PROGRAM MAIN
VAR
	TankControl01				: TankControl;
	Enable						: BOOL;
	TempReq						: REAL := 22.0;
	VolReq						: REAL := 1.2;
	TankDiam					: REAL := 1.0;
	TankHeight					: REAL := 10;
	LevelSensor					: WORD;
	TempSensor					: WORD;
	StartControl				: BOOL;
	FillValve					: BOOL;
	EmptyValve					: BOOL;
	HeatValve					: BOOL;
	
	Temp						: REAL;
	MixerMotor: BOOL;
END_VAR

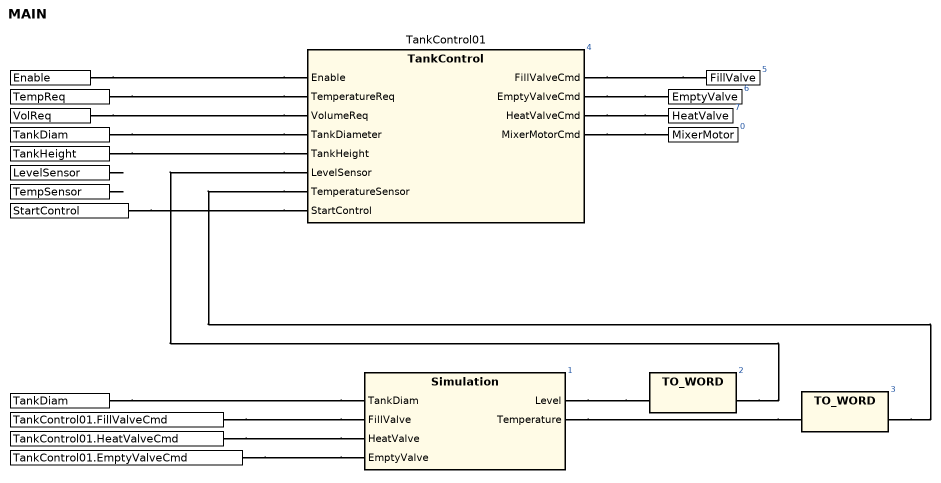
MixerMotor := TankControl01.MixerMotorCmd;
Simulation(TankDiam := TankDiam, FillValve := TankControl01.FillValveCmd, HeatValve := TankControl01.HeatValveCmd, EmptyValve := TankControl01.EmptyValveCmd);
TankControl01(
    Enable := Enable,
    TemperatureReq := TempReq,
    VolumeReq := VolReq,
    TankDiameter := TankDiam,
    TankHeight := TankHeight,
    LevelSensor := TO_WORD(Simulation.Level),
    TemperatureSensor := TO_WORD(Simulation.Temperature),
    StartControl := StartControl); // TankControl
FillValve := TankControl01.FillValveCmd;
EmptyValve := TankControl01.EmptyValveCmd;
HeatValve := TankControl01.HeatValveCmd;
// LevelSensor: input not connected
// TempSensor: input not connected

END_PROGRAM

(* stored: Version 1.1.0.1, ProductVersion 3.1.4024.15
   POU MAIN: Id {8b76ef5a-bbef-48ea-b92b-b61b76f8266b}, SpecialFunc None *)
